(* IEC 61131-3 sources: volt/packages/volt-lsp-iec/test-corpus/lenze-mid/Device/Plc Logic/Application/Library Manager/CmpChecksum, 7 files *)

(* ---- CRC16FINISH.pou ---- *)
FUNCTION CRC16FINISH : WORD
VAR_INPUT
	ULCRC : WORD;
END_VAR
END_FUNCTION

(* ---- CRC16INIT.pou ---- *)
FUNCTION CRC16INIT : WORD
END_FUNCTION

(* ---- CRC16UPDATE.pou ---- *)
FUNCTION CRC16UPDATE : WORD
VAR_INPUT
	ULCRC : WORD;
	PDATA : POINTER TO BYTE;
	ULSIZE : __XWORD;
END_VAR
END_FUNCTION

(* ---- CRC32FINISH.pou ---- *)
FUNCTION CRC32FINISH : DWORD
VAR_INPUT
	ULCRC : DWORD;
END_VAR
END_FUNCTION

(* ---- CRC32INIT.pou ---- *)
FUNCTION CRC32INIT : DWORD
END_FUNCTION

(* ---- CRC32UPDATE.pou ---- *)
FUNCTION CRC32UPDATE : DWORD
VAR_INPUT
	ULCRC : DWORD;
	PDATA : POINTER TO BYTE;
	ULSIZE : __XWORD;
END_VAR
END_FUNCTION

(* ---- CRC32UPDATE2.pou ---- *)
FUNCTION CRC32UPDATE2 : DWORD
VAR_INPUT
	ULCRC : DWORD;
	PDATA : POINTER TO BYTE;
	ULSIZE : __XWORD;
END_VAR
END_FUNCTION
